Fanuc KAREL source: kt00548.KL

-- PROVISIONAL review KL for V1013-1; original PC SHA256 2f75c5cb94684671e9b80bb4399fcec10aa04dd62e25c150cf960cc0b777743a
-- Incomplete behavior may be omitted. Consult companion uncertainty JSON. Do not deploy.
PROGRAM KT00548
%NOLOCKGROUP
VAR
  OUT : BOOLEAN
-- UNRESOLVED_DECL P1 type=000199
-- UNRESOLVED_DECL P2 type=000199
BEGIN
  -- UNRESOLVED_PC offsets 5-38; opcodes 49,7E,49,7E,AC,23
  -- UNRESOLVED_PC offsets 43-47; opcodes 7F
END KT00548
